{attribute 'linkalways'} 
{attribute 'no_explicit_call' := 'This FB is a CLASS and must be accessed using methods or properties'}
{attribute 'enable_dynamic_creation'}
FUNCTION_BLOCK _Array0to9OfITcVnImage EXTENDS ArrayDatatypeBase
VAR CONSTANT
	lBound : DINT := 0;
	uBound : DINT := 9;
END_VAR
VAR
	localData : ARRAY [lBound..uBound] OF ITcVnImage;
	activeData : REFERENCE TO ARRAY [lBound..uBound] OF ITcVnImage REF= localData;
	elements : ARRAY [lBound..uBound] OF _ITcVnImage;
	baseType : _ITcVnImage;
END_VAR

PROPERTY PUBLIC Address : PVOID
GET
Address := ADR(activeData);
END_GET
END_PROPERTY

PROPERTY PUBLIC BaseDatatype : I_Datatype
GET
BaseDatatype := baseType;
END_GET
END_PROPERTY

METHOD PUBLIC ClearReference
VAR_INPUT
END_VAR
activeData REF= localData;
SetElementReference();
END_METHOD

METHOD PUBLIC Clone : I_Datatype
VAR
    pClone : POINTER TO _Array0to9OfITcVnImage;
END_VAR
pClone := __NEW(_Array0to9OfITcVnImage());
pClone^.Value := Value;
Clone := pClone^;
END_METHOD

METHOD FB_init : BOOL
VAR_INPUT
	bInitRetains : BOOL; // if TRUE, the retain variables are initialized (warm start / cold start)
	bInCopyCode : BOOL;  // if TRUE, the instance afterwards gets moved into the copy code (online change)
END_VAR
SetElementReference();
END_METHOD

METHOD PUBLIC GetElementAsDatatypeByIndex : I_Datatype
VAR_INPUT
	Index : DINT;
END_VAR
GetElementAsDatatypeByIndex := elements[Index];
END_METHOD

METHOD PUBLIC GetElementByIndex : REFERENCE TO _ITcVnImage;
VAR_INPUT
	Index : DINT;
END_VAR
GetElementByIndex REF= elements[Index];
END_METHOD

PROPERTY PUBLIC LowerBound : DINT
GET
LowerBound := lBound;
END_GET
END_PROPERTY

METHOD PUBLIC MakeReferenceTo
VAR_INPUT
	ReferenceTarget : REFERENCE TO ARRAY [lBound..uBound] OF ITcVnImage;
END_VAR
activeData REF= ReferenceTarget;
SetElementReference();
END_METHOD

METHOD PROTECTED OnSerializeArrayValues
VAR_INPUT
	Serializer : I_Serializer;
END_VAR
VAR
	i : DINT;
END_VAR
FOR i := lBound TO uBound DO
	elements[i].SerializeWith(Serializer);
END_FOR
END_METHOD

METHOD PROTECTED SetElementReference
VAR_INPUT
END_VAR
VAR
	i : DINT;
END_VAR
FOR i := lBound TO uBound DO
	elements[i].MakeReferenceTo(activeData[i]);
END_FOR
END_METHOD

PROPERTY PUBLIC Size : UDINT
GET
Size := SIZEOF(activeData);
END_GET
END_PROPERTY

METHOD PROTECTED TryDeserializeArrayValues : BOOL
VAR_INPUT
	Deserializer : I_Deserializer;
	Feedback : I_DeserializerFeedback;
END_VAR
VAR
	enumerator : I_DeserializerArrayForwardEnumerator;
	i : DINT;
END_VAR
enumerator := Deserializer.GetArrayEnumerator();
i := lBound;

WHILE enumerator.MoveNext() AND i <= uBound DO
	
	IF NOT elements[i].TryDeserializeFrom(enumerator.Current, Feedback) THEN
		EXIT;
	END_IF
	i := i + 1;

END_WHILE
enumerator.Dispose();
END_METHOD

METHOD TryMakeReferenceTo : BOOL
VAR_INPUT
	Target : I_Datatype;
END_VAR
VAR
	targetAsArray : I_ArrayDatatype;
	pTargetData : POINTER TO ARRAY [lBound..uBound] OF ITcVnImage;
END_VAR
IF NOT Target.TryResolveAsArrayDatatype(targetAsArray) THEN
	RETURN;
END_IF

IF NOT (targetAsArray.Identifier = Identifier) THEN
	RETURN;
END_IF

pTargetData := Target.Address;
activeData REF= pTargetData^;
SetElementReference();
TryMakeReferenceTo := TRUE;
END_METHOD

PROPERTY PUBLIC UpperBound : DINT
GET
UpperBound := ubound;
END_GET
END_PROPERTY

PROPERTY PUBLIC Value : REFERENCE TO ARRAY [lBound..uBound] OF ITcVnImage;
GET
Value ref= activeData;
END_GET
END_PROPERTY

END_FUNCTION_BLOCK

(* stored: Version 1.1.0.1, ProductVersion 3.1.4024.13
   POU _Array0to9OfITcVnImage: Id {53378396-ddd0-01d6-1fe9-e5bade8d0852}, SpecialFunc None
   Folder Core: Id {ee370253-d404-08ac-12f9-cbf2a99a050f}
   Folder Constructor: Id {62b372c4-481f-04c0-3753-6725e42e3748}
   Folder Protected: Id {ee2c7fe3-2ae9-0189-3b2a-465e80ce9a73}
   Folder Customize: Id {6082933d-8e3c-03d6-17ac-83eed2eb385f}
   Property Address: Id {b1798d1e-082e-09a9-0d37-cf8b71fd7433}
   Get Get: Id {52610a41-1e81-05e2-2691-b1b5f19e6184}
   Property BaseDatatype: Id {03ef3308-5246-05a4-1de8-25637cc4f48b}
   Get Get: Id {c04feab5-77b2-0bdd-1109-9d17214e2cd7}
   Method ClearReference: Id {cd1df7c2-9ccb-022f-3224-2a649fbe2d54}
   Method Clone: Id {a45e0e84-1483-0d52-2184-26fe9c42b26e}
   Method FB_init: Id {3ff5896f-35b4-0a53-205a-62107e076d42}
   Method GetElementAsDatatypeByIndex: Id {a9fb7e81-a741-073c-2a6b-1df33bc866fd}
   Method GetElementByIndex: Id {34e801df-5fc2-0acf-2118-b20a89c11d37}
   Property LowerBound: Id {3511022f-6cfb-0308-2ebe-140c019ada94}
   Get Get: Id {7e67209e-af8b-07d1-0b68-2b63fa5b7433}
   Method MakeReferenceTo: Id {679eb237-e4c1-0b1d-271a-f2529878e181}
   Method OnSerializeArrayValues: Id {4e82bd63-664a-0eef-08dc-6bce4a0d8f32}
   Method SetElementReference: Id {d2bba348-755f-0edc-31ab-dc63b9a7feb6}
   Property Size: Id {7be66c13-ce8f-0df0-3e98-dc3c15dfd88a}
   Get Get: Id {bcac942a-1bab-0433-1e66-4b0a9a729af9}
   Method TryDeserializeArrayValues: Id {79cb0502-d0fb-0d0b-34a9-441464dbd035}
   Method TryMakeReferenceTo: Id {e540e74c-b883-0bc0-2019-6dd7114ce613}
   Property UpperBound: Id {13e3a5dc-2917-05ba-1344-b4f240534732}
   Get Get: Id {26dbe2aa-17ab-01f9-1dbf-a58ee37e3620}
   Property Value: Id {96672d1c-be7f-0582-2f79-66e8b61430a4}
   Get Get: Id {68fe547c-9461-01fe-01f1-6ee341c80324} *)
